Staubli VAL3: moveHome.pgx

program moveHome()
begin
  movej(homePosition,flange,mFastMov)
  waitEndMove()
  message="moveHome:done"
  taskCreate "sendStatus",100,sendStatus()
  taskKill("moveHome")
end
